{attribute 'qualified_only'}
{attribute 'strict'}
TYPE
    eTagPairingStatus :
    (
        Unknown := 0,
        Active := 10,
        Inactive := 20
    );
END_TYPE

(* stored: Version 1.1.0.1
   DUT eTagPairingStatus: Id {2c9e8f95-d8ce-40d9-9a51-484b94116cb3} *)
